ADAPTER IEmergencyPhase (* Adapter Interface *)
  (* Standard: 61499-1 *)
  (* Version 0.0, 7/6/2026, Schneider Electric *)
  PACKAGE SE.Nereda;
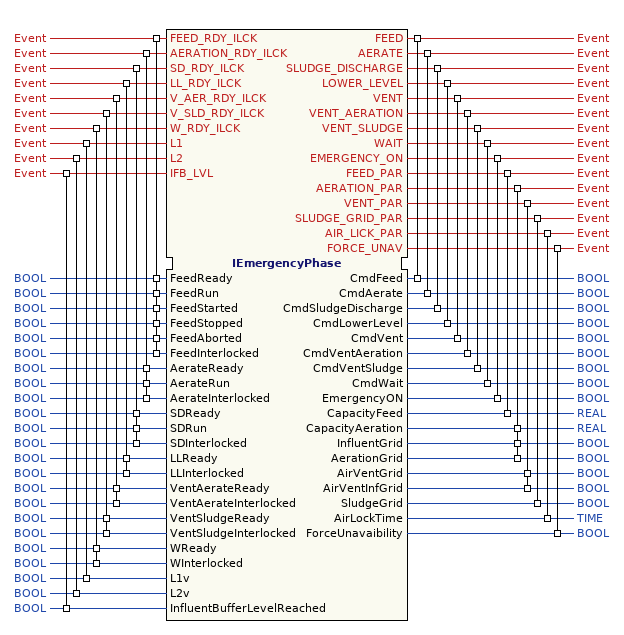
  EVENT_INPUT
    FEED_RDY_ILCK WITH FeedReady, FeedRun, FeedStarted, FeedStopped, FeedAborted, FeedInterlocked;
    AERATION_RDY_ILCK WITH AerateReady, AerateInterlocked, AerateRun;
    SD_RDY_ILCK WITH SDReady, SDInterlocked, SDRun;
    LL_RDY_ILCK WITH LLReady, LLInterlocked;
    V_AER_RDY_ILCK WITH VentAerateReady, VentAerateInterlocked;
    V_SLD_RDY_ILCK WITH VentSludgeReady, VentSludgeInterlocked;
    W_RDY_ILCK WITH WReady, WInterlocked;
    L1 WITH L1v;
    L2 WITH L2v;
    IFB_LVL WITH InfluentBufferLevelReached;
  END_EVENT
  EVENT_OUTPUT
    FEED WITH CmdFeed;
    AERATE WITH CmdAerate;
    SLUDGE_DISCHARGE WITH CmdSludgeDischarge;
    LOWER_LEVEL WITH CmdLowerLevel;
    VENT WITH CmdVent;
    VENT_AERATION WITH CmdVentAeration;
    VENT_SLUDGE WITH CmdVentSludge;
    WAIT WITH CmdWait;
    EMERGENCY_ON WITH EmergencyON;
    FEED_PAR WITH CapacityFeed;
    AERATION_PAR WITH CapacityAeration, InfluentGrid, AerationGrid;
    VENT_PAR WITH AirVentGrid, AirVentInfGrid;
    SLUDGE_GRID_PAR WITH SludgeGrid;
    AIR_LICK_PAR WITH AirLockTime;
    FORCE_UNAV WITH ForceUnavaibility;
  END_EVENT
  VAR_INPUT
    FeedReady : BOOL;
    FeedRun : BOOL;
    FeedStarted : BOOL;
    FeedStopped : BOOL;
    FeedAborted : BOOL;
    FeedInterlocked : BOOL;
    AerateReady : BOOL;
    AerateRun : BOOL;
    AerateInterlocked : BOOL;
    SDReady : BOOL;
    SDRun : BOOL;
    SDInterlocked : BOOL;
    LLReady : BOOL;
    LLInterlocked : BOOL;
    VentAerateReady : BOOL;
    VentAerateInterlocked : BOOL;
    VentSludgeReady : BOOL;
    VentSludgeInterlocked : BOOL;
    WReady : BOOL;
    WInterlocked : BOOL;
    L1v : BOOL;
    L2v : BOOL;
    InfluentBufferLevelReached : BOOL;
  END_VAR
  VAR_OUTPUT
    CmdFeed : BOOL;
    CmdAerate : BOOL;
    CmdSludgeDischarge : BOOL;
    CmdLowerLevel : BOOL;
    CmdVent : BOOL;
    CmdVentAeration : BOOL;
    CmdVentSludge : BOOL;
    CmdWait : BOOL;
    EmergencyON : BOOL;
    CapacityFeed : REAL;
    CapacityAeration : REAL;
    InfluentGrid : BOOL;
    AerationGrid : BOOL;
    AirVentGrid : BOOL;
    AirVentInfGrid : BOOL;
    SludgeGrid : BOOL;
    AirLockTime : TIME;
    ForceUnavaibility : BOOL;
  END_VAR
  SERVICE SOCKET/PLUG
    SEQUENCE request_confirm
      SOCKET.REQ(REQD) -> PLUG.REQ(REQD);
      PLUG.CNF(CNFD) -> SOCKET.CNF(CNFD);
    END_SEQUENCE
    SEQUENCE indication_response
      PLUG.IND(INDD) -> SOCKET.IND(INDD);
      SOCKET.RSP(RSPD) -> PLUG.RSP(RSPD);
    END_SEQUENCE
  END_SERVICE
END_ADAPTER
